{attribute 'GeneratedUsingTerminal: EL1502--0000'}
{attribute addProperty BoxType "EL1502--0000"}
{attribute addProperty Id "Enable_output_functionsAT %Q*BOOL1Set_outputAT %Q*BOOL1Set_counterAT %Q*BOOL1Inhibit_counterAT %Q*BOOL1Set_counter_valueAT %Q*UDINT4"}
{attribute addProperty CRC "3943999093"}
{attribute addProperty Size "8"}
TYPE CNT_Outputs_EB14A675 EXTENDS OutputBase_10CEE7DE :
STRUCT
	{attribute addProperty Name "Enable_output_functions"}
	Enable_output_functions AT %Q* : BOOL;
	{attribute addProperty Name "Set_output"}
	Set_output AT %Q* : BOOL;
	{attribute addProperty Name "Set_counter"}
	Set_counter AT %Q* : BOOL;
	{attribute addProperty Name "Inhibit_counter"}
	Inhibit_counter AT %Q* : BOOL;
	{attribute addProperty Name "Set_counter_value"}
	Set_counter_value AT %Q* : UDINT;
END_STRUCT
END_TYPE

(* stored: Version 1.2.0.0, ProductVersion 3.1.4024.9
   DUT CNT_Outputs_EB14A675: Id {8b2f7c1a-3ed5-46c9-b6c9-0b147b53fe24} *)
